TYPE MC_COMMAND_REF :
STRUCT
	CommandId : INT;
END_STRUCT
END_TYPE

(* stored: Version 1.1.0.1, ProductVersion 3.1.4024.12
   DUT MC_COMMAND_REF: Id {e0495532-0bd3-4a48-9b5f-86251b53fbda} *)
